FUNCTION Matrix_Transpose : Bool
VAR_IN_OUT CONSTANT
	M_From : Matrix;
END_VAR
VAR_IN_OUT
	M_To : Matrix;
END_VAR
VAR
	Ri : UINT;
	Ci : UINT;
END_VAR

IF M_From.Rows <> M_To.Cols OR M_From.Cols <> M_to.Rows THEN
	Matrix_Transpose := FALSE;
	RETURN;
END_IF

Matrix_Transpose := TRUE;

FOR Ri := 0 TO M_From.Rows-1 DO
	FOR Ci := 0 TO M_From.Cols-1 DO
		M_To.SetRC(Ci,Ri,M_From.GetRC(Ri,Ci));
	END_FOR
END_FOR

END_FUNCTION

(* stored: Version 1.1.0.1, ProductVersion 3.1.4024.9
   POU Matrix_Transpose: Id {9e8611eb-e7e8-49d4-8541-b23bf7999d2e}, SpecialFunc None *)
